{attribute 'qualified_only'}
{attribute 'strict'}
TYPE CmdActuator :
(
	None,
	Extend,
	Retract,
	Reset
);
END_TYPE

(* stored: Version 1.1.0.1, ProductVersion 3.1.4022.11
   DUT CmdActuator: Id {e3044dd0-7f55-4203-a6ea-e1e1cf0b94c8} *)
